FUNCTION_BLOCK PrecargaLiqInyeccion
VAR_INPUT
	CaudalimetroSup:REAL;
	Precarga:BOOL;
	VeloBombaSolicitada:REAL;
END_VAR
VAR_OUTPUT
	MarchaBomba:BOOL;
	VelocidadBomba:REAL;
END_VAR
VAR
END_VAR

IF CaudalimetroSup<0 THEN
	MarchaBomba:=TRUE;
	ELSE
	MarchaBomba:=FALSE;	
END_IF

END_FUNCTION_BLOCK

(* stored: Version 1.1.0.1, ProductVersion 3.1.4024.12
   POU PrecargaLiqInyeccion: Id {ae542e02-1f0f-402b-9006-94a38496e16c}, SpecialFunc None *)
